// Implicitly generated code : DO NOT EDIT
FUNCTION CheckDivLInt : LINT
VAR_INPUT
	divisor:LINT;
END_VAR

// Implicitly generated code: Only an implementation suggestion
{noflow}
IF divisor = 0 THEN
	CheckDivLInt:=1;
ELSE
	CheckDivLInt:=divisor;
END_IF;

END_FUNCTION

(* stored: Version 1.1.0.1, ProductVersion 3.1.4026.8
   POU CheckDivLInt: Id {6ad22c91-29f5-4808-9b6e-302f12bb99c5}, SpecialFunc CheckDivInt64 *)
